FUNCTION_BLOCK BaseTestSuite
VAR_INPUT
END_VAR
VAR_OUTPUT
END_VAR
VAR
END_VAR

END_FUNCTION_BLOCK

(* stored: Version 1.1.0.1
   POU BaseTestSuite: Id {92552d02-200d-47eb-ae91-d0e3f8621688}, SpecialFunc None *)
